SUBAPPLICATION GreenWhiteBackground_Heckschieber (* Subapplication Type *)
  (* Standard: 61499-2 *)
  (* Version 1.0, 2023-02-11, franz *)
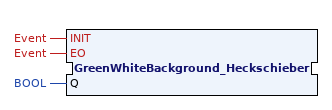
  EVENT_INPUT
    INIT;
    EO;
  END_EVENT
  VAR_INPUT
    Q : BOOL;
  END_VAR
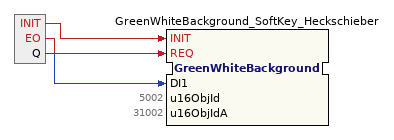
  FBS
    GreenWhiteBackground_SoftKey_Heckschieber : GreenWhiteBackground(u16ObjId := 5002, u16ObjIdA := 31002);
  END_FBS
  EVENT_CONNECTIONS
    INIT TO GreenWhiteBackground_SoftKey_Heckschieber.INIT;
    EO TO GreenWhiteBackground_SoftKey_Heckschieber.REQ;
  END_CONNECTIONS
  DATA_CONNECTIONS
    Q TO GreenWhiteBackground_SoftKey_Heckschieber.DI1;
  END_CONNECTIONS
END_SUBAPPLICATION
